PROGRAM MAIN
VAR
END_VAR

END_PROGRAM

(* stored: Version 1.1.0.1
   POU MAIN: Id {8446e5cd-71d3-4dbf-a2dd-a38b81fd53ce} *)
